# EPICS substitutions: iocBoot/iocLinux/asynRecord.substitutions
file "$(ASYN)/db/asynRecord.db"
{
pattern
{P        R         PORT    ADDR    OMAX  IMAX}
{xxx:     asyn_1   serial1    0     256  256}
{xxx:     asyn_2   serial2    0     256  256}
{xxx:     asyn_3   serial3    0     256  256}
{xxx:     asyn_4   serial4    0     256  256}
}
